{attribute addProperty BoxType "EK1100-0000-0018"}
{attribute addProperty Id "Beckhoff_EP5xxxEK1122Beckhoff_EP5xxxEK1122_413134381928241"}
{attribute addProperty CRC "2410141296"}
{attribute addProperty SizeInBites "1928"}
{attribute addProperty SizeInBytes "241"}
TYPE Beckhoff_EP5xxx_8FA7D670 EXTENDS EK1100_179A0949 :
STRUCT
	{attribute addProperty Name "Beckhoff_EP5xxxEK1122"}
	Beckhoff_EP5xxxEK1122 : Beckhoff_EP5xxxEK1122_41313438;
END_STRUCT
END_TYPE

(* stored: Version 1.2.0.0, ProductVersion 3.1.4024.9
   DUT Beckhoff_EP5xxx_8FA7D670: Id {40acb0e9-1630-4aca-bc93-667312e5c526} *)
